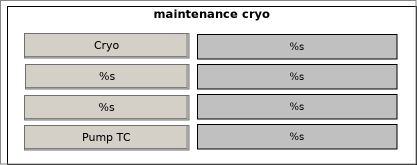
VISUALIZATION VISU_MAINT_CRYO_AC  // 417x165
VAR_IN_OUT
	COM: BLOCK_RS232_ONBOARD_V4;
END_VAR
    RoundedRectangle (7,6 410x159), "maintenance cryo", text list: 'TextList_CryoPump', text index: 97
    Rectangle (197,34 200x25), "%s", text variable: COM.PRM_PumpStartDelay, text list: 'TextList_CryoPump', text index: BOOL_TO_INT(COM.STATE_Pompe)+7
    Rectangle (197,64 200x25), "%s", text list: 'TextList_CryoPump', text index: BOOL_TO_INT(COM.STATE_Rough_valve)+37
    Rectangle (197,94 200x25), "%s", text list: 'TextList_CryoPump', text index: BOOL_TO_INT(COM.STATE_Purge_valve)+37
    Button (24,33 165x25), "Cryo"
        OnMouseClick: execute {
            IF (COM.CO_Etat=TRUE) THEN
            	com.CO_Etat:=FALSE;
            ELSE
            	com.CO_Etat:=TRUE;
            END_IF
        }
    Button (25,64 164x25), "%s", text list: 'TextList_CryoPump', text index: 41
        OnMouseClick: execute {
            IF (COM.CO_RoughValve=TRUE) THEN
            	com.CO_RoughValve:=FALSE;
            ELSE
            	com.CO_RoughValve:=TRUE;
            END_IF
        }
    Button (24,95 165x25), "%s", text list: 'TextList_CryoPump', text index: 42
        OnMouseClick: execute {
            IF (COM.CO_PurgeValve=TRUE) THEN
            	com.CO_PurgeValve:=FALSE;
            ELSE
            	com.CO_PurgeValve:=TRUE;
            END_IF
        }
    Rectangle (197,124 200x25), "%s", text list: 'TextList_CryoPump', text index: BOOL_TO_INT(COM.STATE_Pump_TC)
    Button (24,125 165x25), "Pump TC"
        OnMouseClick: execute {
            IF (COM.CO_PumpTc=TRUE) THEN
            	com.CO_PumpTc:=FALSE;
            ELSE
            	com.CO_PumpTc:=TRUE;
            END_IF
        }
END_VISUALIZATION

(* stored: Version 1.1.0.1, ProductVersion 3.1.4026.18
   Visu VISU_MAINT_CRYO_AC: Id {6be7c0f5-637c-49bf-a1c6-a311bad1d35d} *)
